PROGRAM Heraus_Heater_Control

VAR_INPUT
		HMI_RECIPE_NUM : INT; // SELECTED RECIPE VALUE FROM HMI NUMERIC INPUT
		
		HERAUS_STATUS  : INT; // BINARY STATUS INFORMATION FROM HEATER CABINET.
							  // 0 = OFF
							  // 1 = SYSTEM STARTING
							  // 2 = POST HEATING GAS ON
							  // 3 = RUNNING
							  // 4 = STANDBY
END_VAR

VAR
	HERAUS_ESTOP_OK      AT %I*: BOOL; // ESTOP OK INTERLOCK RELAY STATE
	HERAUS_STATUS_B1     AT %I*: BOOL; // HEARAUS HEATER STATUS BIT 1
	HERAUS_STATUS_B2     AT %I*: BOOL; // HEARAUS HEATER STATUS BIT 2
	HERAUS_STATUS_B3     AT %I*: BOOL; // HEARAUS HEATER STATUS BIT 3
	RECIPE_VALUE_BIT_0   AT %Q*: BOOL; // BINARY VALUE 1 RECIPE SELECTION
	RECIPE_VALUE_BIT_1   AT %Q*: BOOL; // BINARY VALUE 2 RECIPE SELECTION
	RECIPE_VALUE_BIT_2   AT %Q*: BOOL; // BINARY VALUE 4 RECIPE SELECTION
	RECIPE_VALUE_BIT_3   AT %Q*: BOOL; // BINARY VALUE 8 RECIPE SELECTION
	RECIPE_VALUE_BIT_4   AT %Q*: BOOL; // BINARY VALUE 16 RECIPE SELECTION
		
END_VAR

// INITIALIZE HEATER STATUS TO 0
		HERAUS_STATUS := 0;
IF HERAUS_STATUS_B1 AND NOT HERAUS_STATUS_B2 AND NOT HERAUS_STATUS_B3 THEN
		HERAUS_STATUS := 1;
ELSIF HERAUS_STATUS_B2 AND NOT HERAUS_STATUS_B1 AND NOT HERAUS_STATUS_B3 THEN
		HERAUS_STATUS := 2;
ELSIF HERAUS_STATUS_B3 AND NOT HERAUS_STATUS_B1 AND NOT HERAUS_STATUS_B2 THEN
		HERAUS_STATUS := 3;
ELSIF HERAUS_STATUS_B3 AND HERAUS_STATUS_B1 AND NOT HERAUS_STATUS_B2 THEN
		HERAUS_STATUS := 4;
END_IF

CASE HMI_RECIPE_NUM OF 
     1 : RECIPE_VALUE_BIT_0 := TRUE; 
         RECIPE_VALUE_BIT_1 := FALSE; 
		 RECIPE_VALUE_BIT_2 := FALSE;
		 RECIPE_VALUE_BIT_3 := FALSE;
		 RECIPE_VALUE_BIT_4 := FALSE; 

     2 : RECIPE_VALUE_BIT_0 := FALSE; 
         RECIPE_VALUE_BIT_1 := TRUE;
		 RECIPE_VALUE_BIT_2 := FALSE;
		 RECIPE_VALUE_BIT_3 := FALSE;
		 RECIPE_VALUE_BIT_4 := FALSE; 

	 3 : RECIPE_VALUE_BIT_0 := TRUE; 
         RECIPE_VALUE_BIT_1 := TRUE;
		 RECIPE_VALUE_BIT_2 := FALSE;
		 RECIPE_VALUE_BIT_3 := FALSE;
		 RECIPE_VALUE_BIT_4 := FALSE; 
		 
	 4 : RECIPE_VALUE_BIT_0 := FALSE; 
         RECIPE_VALUE_BIT_1 := FALSE;
		 RECIPE_VALUE_BIT_2 := TRUE;
		 RECIPE_VALUE_BIT_3 := FALSE;
		 RECIPE_VALUE_BIT_4 := FALSE; 
		 
	 5 : RECIPE_VALUE_BIT_0 := TRUE; 
         RECIPE_VALUE_BIT_1 := FALSE;
		 RECIPE_VALUE_BIT_2 := TRUE;
		 RECIPE_VALUE_BIT_3 := FALSE;
		 RECIPE_VALUE_BIT_4 := FALSE; 

     6 : RECIPE_VALUE_BIT_0 := FALSE; 
         RECIPE_VALUE_BIT_1 := TRUE;
		 RECIPE_VALUE_BIT_2 := TRUE;
		 RECIPE_VALUE_BIT_3 := FALSE;
		 RECIPE_VALUE_BIT_4 := FALSE; 

	 7 : RECIPE_VALUE_BIT_0 := TRUE; 
         RECIPE_VALUE_BIT_1 := TRUE;
		 RECIPE_VALUE_BIT_2 := TRUE;
		 RECIPE_VALUE_BIT_3 := FALSE;
		 RECIPE_VALUE_BIT_4 := FALSE; 
		 
	 8 : RECIPE_VALUE_BIT_0 := FALSE; 
         RECIPE_VALUE_BIT_1 := FALSE;
		 RECIPE_VALUE_BIT_2 := FALSE;
		 RECIPE_VALUE_BIT_3 := TRUE;
		 RECIPE_VALUE_BIT_4 := FALSE; 
		 
	 9 : RECIPE_VALUE_BIT_0 := TRUE; 
         RECIPE_VALUE_BIT_1 := FALSE;
		 RECIPE_VALUE_BIT_2 := FALSE;
		 RECIPE_VALUE_BIT_3 := TRUE;
		 RECIPE_VALUE_BIT_4 := FALSE; 
		 
	10 : RECIPE_VALUE_BIT_0 := FALSE; 
         RECIPE_VALUE_BIT_1 := TRUE;
		 RECIPE_VALUE_BIT_2 := FALSE;
		 RECIPE_VALUE_BIT_3 := TRUE;
		 RECIPE_VALUE_BIT_4 := FALSE; 
		
ELSE 
	     RECIPE_VALUE_BIT_0 := FALSE; 
         RECIPE_VALUE_BIT_1 := FALSE;
		 RECIPE_VALUE_BIT_2 := FALSE;
		 RECIPE_VALUE_BIT_3 := FALSE;
		 RECIPE_VALUE_BIT_4 := FALSE; 
END_CASE;

END_PROGRAM

(* stored: Version 1.1.0.1, ProductVersion 3.1.4024.12
   POU Heraus_Heater_Control: Id {9435777a-9821-4d70-8036-dc6683a37a24}, SpecialFunc None *)
